// TIA Portal V18 export
// export: Created 2026-06-08T17:01:58.4505211Z, ExportSetting WithDefaults, DisplayName Totally Integrated Automation Portal, DisplayVersion V18, DisplayName TIA Portal Openness, DisplayVersion V18, DisplayName TIA Portal Version Control Interface, DisplayVersion V18, DisplayName STEP 7 Professional, DisplayVersion V18, DisplayName STEP 7 Safety, DisplayVersion V18, DisplayName WinCC Professional, DisplayVersion V18
FUNCTION_BLOCK "M1_MOTOR"   // FB2, LAD
{ S7_Optimized_Access := 'TRUE' }
VERSION : 0.1
// stored: AutoNumber true, IsIECCheckEnabled false, IsRetainMemResEnabled false, MemoryReserve 100, SetENOAutomatically false, UDAEnableTagReadback false
   VAR_INPUT
      EMERGENCY_STATE : Bool;
      WIND_DOWN : Bool;
      INTERLOCK_R : Bool;
      MOVE_R : Bool;
      INTERLOCK_F : Bool;
      MOVE_F : Bool;
      COIL_F : Bool;
      TRIP_COUNT_FINISHED : Bool;
   END_VAR
   VAR_OUTPUT
      COIL_R_OUT : Bool;
      COIL_R_OUT_HMI : Bool;
      COIL_F_OUT : Bool;
      COIL_F_OUT_HMI : Bool;
   END_VAR
BEGIN

REGION Network 1
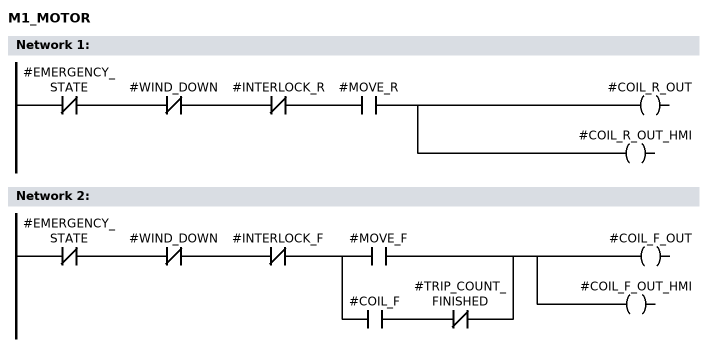
   RUNG wire#powerrail
      I_Contact( #EMERGENCY_STATE )
      I_Contact( #WIND_DOWN )
      I_Contact( #INTERLOCK_R )
      Contact( #MOVE_R )
      wire#w1
      Coil( #COIL_R_OUT )
   END_RUNG
   RUNG wire#w1
      Coil( #COIL_R_OUT_HMI )
   END_RUNG
   // the same network as SCL:
   #COIL_R_OUT := NOT #EMERGENCY_STATE AND NOT #WIND_DOWN AND NOT #INTERLOCK_R AND #MOVE_R;
   #COIL_R_OUT_HMI := #COIL_R_OUT;
END_REGION

REGION Network 2
   RUNG wire#powerrail
      I_Contact( #EMERGENCY_STATE )
      I_Contact( #WIND_DOWN )
      I_Contact( #INTERLOCK_F )
      wire#w1
      Contact( #MOVE_F )
      wire#w2
      Coil( #COIL_F_OUT )
   END_RUNG
   RUNG wire#w1
      Contact( #COIL_F )
      I_Contact( #TRIP_COUNT_FINISHED )
   END_RUNG wire#w2
   RUNG wire#w2
      Coil( #COIL_F_OUT_HMI )
   END_RUNG
   // the same network as SCL:
   #COIL_F_OUT := NOT #EMERGENCY_STATE AND NOT #WIND_DOWN AND NOT #INTERLOCK_F AND (#MOVE_F OR (#COIL_F AND NOT #TRIP_COUNT_FINISHED));
   #COIL_F_OUT_HMI := #COIL_F_OUT;
END_REGION
END_FUNCTION_BLOCK
